FUNCTION_BLOCK SignalTimeRecorder
VAR_INPUT
END_VAR
VAR_OUTPUT
END_VAR
VAR
  _record_delay: TIME;
  _signal: BOOL;
  _duration_on: TIME;
  _duration_off: TIME;
  _signal_filtertime: TIME;
  filtertime: TIME;
  t_record_delay: TON;
END_VAR

PROPERTY duration_off : TIME
GET
duration_off := _duration_off;
END_GET
END_PROPERTY

PROPERTY duration_on : TIME
GET
duration_on := _duration_on;
END_GET
END_PROPERTY

PROPERTY off_ratio : REAL
GET
off_ratio := 1.0 - on_ratio;
END_GET
END_PROPERTY

PROPERTY on_ratio : REAL
GET
IF (record_duration = T#0S) THEN
  on_ratio := TO_REAL(signal);
ELSE
  on_ratio := TO_REAL(duration_on) / TO_REAL(record_duration);
END_IF
END_GET
END_PROPERTY

METHOD record
VAR_INPUT
  execute: BOOL;
END_VAR
VAR
  act_timestamp: TIME;
  previous_cycle_time: TIME;
END_VAR
VAR_INST
  r_execute: R_TRIG;
  previous_timestamp: TIME;
  t_signal_filtertime: TON;
END_VAR
t_record_delay(IN:=execute, PT:=record_delay);
r_execute(CLK:=execute);
IF r_execute.Q THEN
  _duration_on := T#0S;
  _duration_off := T#0S;
  filtertime := T#0S;
  previous_timestamp := T#0S;
END_IF

IF t_record_delay.Q THEN
  act_timestamp := GetSystemTimeAsTime();
  
  IF previous_timestamp = T#0S THEN
    previous_cycle_time := T#0S;
  ELSE
    previous_cycle_time := act_timestamp - previous_timestamp;
  END_IF
  previous_timestamp := act_timestamp;
  
  t_signal_filtertime(IN:=signal, PT:=signal_filtertime);
  IF t_signal_filtertime.Q AND (filtertime > T#0S) THEN
    _duration_on := _duration_on + filtertime;
    filtertime := T#0S;
    _duration_on := _duration_on + previous_cycle_time;
  ELSIF t_signal_filtertime.Q THEN
    _duration_on := _duration_on + previous_cycle_time;
  ELSIF NOT t_signal_filtertime.Q AND signal THEN
    filtertime := filtertime + previous_cycle_time;
  ELSIF NOT signal AND (filtertime > T#0S) THEN
    _duration_off := _duration_off + filtertime;
    filtertime := T#0S;
    _duration_off := _duration_off + previous_cycle_time;
  ELSE
    _duration_off := _duration_off + previous_cycle_time;
  END_IF
END_IF
END_METHOD

PROPERTY record_delay : TIME
GET
record_delay := _record_delay;
END_GET
SET
_record_delay := record_delay;
END_SET
END_PROPERTY

PROPERTY record_duration : TIME
GET
record_duration := duration_on + duration_off;
END_GET
END_PROPERTY

METHOD reset
VAR_INPUT
END_VAR
_duration_off := T#0S;
_duration_on := T#0S;
END_METHOD

PROPERTY signal : BOOL
GET
signal := _signal;
END_GET
SET
_signal := signal;
END_SET
END_PROPERTY

PROPERTY signal_filtertime : TIME
GET
signal_filtertime := _signal_filtertime;
END_GET
SET
_signal_filtertime := signal_filtertime;
END_SET
END_PROPERTY

PROPERTY started_recording : BOOL
GET
started_recording := t_record_delay.Q;
END_GET
END_PROPERTY

END_FUNCTION_BLOCK

(* stored: Version 1.1.0.1, ProductVersion 3.1.4022.18
   POU SignalTimeRecorder: Id {50b9ef85-d5ef-4f95-8c90-21444817cbcb}, SpecialFunc None
   Property duration_off: Id {3c86d980-0079-4474-8f55-4dfb55305b84}
   Get Get: Id {915b8f38-c90b-4109-a1f0-106263406f3e}
   Property duration_on: Id {faf4f117-4bff-46ef-a2d4-1b939b6cd0af}
   Get Get: Id {fcde13a2-5eb8-4d10-ae73-46a50e964b20}
   Property off_ratio: Id {85048ccd-8de4-4fb6-b9e5-98cd3fb800db}
   Get Get: Id {a5c26eaa-980c-4a8c-8005-0adb65deebf5}
   Property on_ratio: Id {ececa6fb-d525-4ab0-8b9f-868e0e7bc108}
   Get Get: Id {ba7ec5d4-cced-42da-9b31-a4ec08edab63}
   Method record: Id {42cca3e1-0f64-43a6-b22d-a3f0f91c42a0}
   Property record_delay: Id {95d9a1c4-8e87-46ed-8d04-bc53f705999a}
   Get Get: Id {3bb3a519-2cce-436a-8759-3baf23b886ee}
   Set Set: Id {f025a2f7-3ef3-4af8-a769-e8995ed0180c}
   Property record_duration: Id {319c6fb6-8e66-404e-81b2-83e5cc05d8a8}
   Get Get: Id {33191238-4f76-4ba7-9e9b-b18ff5e65f36}
   Method reset: Id {403d21f2-b5c3-4dc4-ab80-2046b11e0d45}
   Property signal: Id {2394856c-94b8-49e0-b910-cfaded13c1c4}
   Get Get: Id {25559d9c-83ee-45db-905b-2b628ba87e46}
   Set Set: Id {16fc0461-a034-415d-bf77-d87535d83777}
   Property signal_filtertime: Id {3a9d6243-6894-4561-bffb-ab8d019d4d69}
   Get Get: Id {79943585-e570-46cb-8d8e-87dd48995671}
   Set Set: Id {3f6b2ae9-e3bc-4a5c-acc9-3b8b545b7ffb}
   Property started_recording: Id {7c4c7628-eef1-429e-b9ba-7339a0728161}
   Get Get: Id {21a601a3-ad4e-4484-b2a4-a435869c88d1} *)
